Fanuc KAREL source: DAQ_CHECKP.kl

PROGRAM T
%NOLOCKGROUP
VAR
 v0 : INTEGER
 v1 : INTEGER
 v2 : INTEGER
BEGIN
 DAQ_CHECKP(v0, v1, v2)
END T
